// SIMATIC S7-200 project (STEP 7-Micro/WIN), CPU 221 REL 01.10

SYMBOL_TABLE USR1
First_Scan_On    SM0.1    // This bit is on for the first scan cycle only.
Edge_Up          MW1      // The number of positive transitions at input I0.0 is stored in MW1.
Edge_Down        MW3      // The number of negative transitions at input I0.1 is stored in MW3.
END_SYMBOL_TABLE

ORGANIZATION_BLOCK MAIN:OB1
TITLE=
//  题目：检测输入信号的边沿
// ***概述***
// 本例程序用来说明如何用S7-200的检测边沿指令来检测简单信号的变化。在这个过程中，
// 用上升和下降来区分信号边沿，上升沿指信号由“0”变为“1”，下降沿指信
// 号由“1”变为“0”。逻辑“1”表示输入上有电压，“0”表示输入上无电压。
// 程序用2个存储字分别累计输入I0.0上升沿数目以及输入I0.1下降沿数目。
// ***程序和注释***
// 程序例用输入I0.0和EU（上升沿）指令来判定上升沿变化是否发生，也就是说，
// 信号由“0”变为“1”。如果一个上升沿变化发生了，那么存储字MW1的值增加1
// ED(下降沿)指令用来计数输入I0.1的下降沿，用存储字MW3来计数。如果某一个
// 存储字计数达到127，那么该存储字被重新置为0。注意MB2是存储字MW1的低字节，
// MB1为高字节。同样的，MB4为存储字MW3的低字节，MB3为高字节。
// 标题：检测边沿
// 
BEGIN
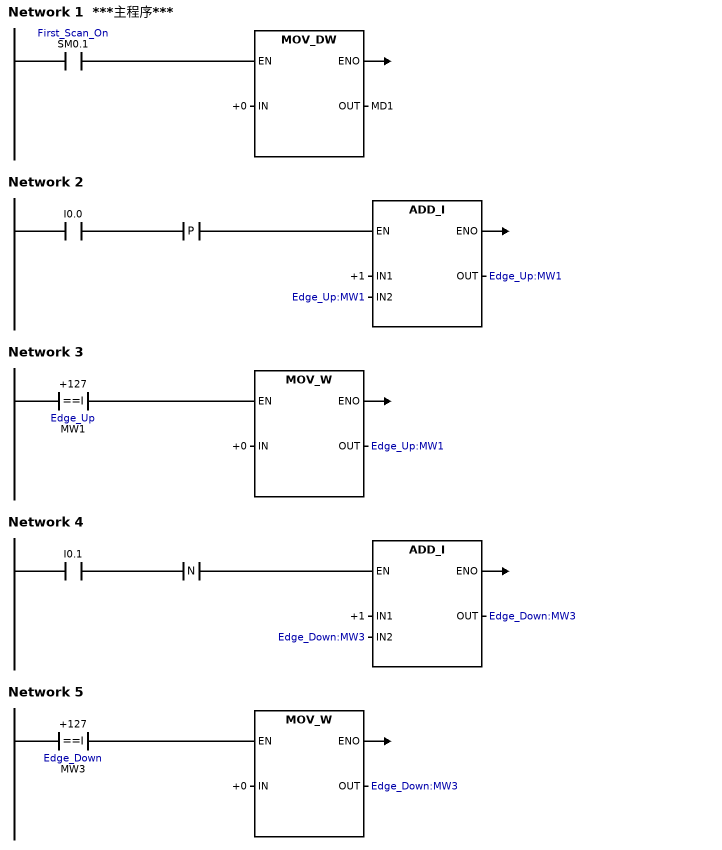
Network 1 // ***主程序***	
// 仅在第一次扫描时 SM0.1=1。
// 把存储器双字 MD1置0
LD     First_Scan_On:SM0.1
MOVD   +0, MD1
Network 2
// 输入信号 I0.0.
// 上升沿
// 存储字MW1的值加1
LD     I0.0
EU
+I     +1, Edge_Up:MW1
Network 3
// 如果累计127个上升沿变化（或某个指定的值）
// 则将存储字MW1置0
LDW=   +127, Edge_Up:MW1
MOVW   +0, Edge_Up:MW1
Network 4
// 输入信号 I0.0.
// 下降沿
// 下降沿变化，使存储字MW3的值加1
LD     I0.1
ED
+I     +1, Edge_Down:MW3
Network 5
// 如果累计127个下降沿变化（或某个指定的值）
//则将存储字MW3置0
LDW=   +127, Edge_Down:MW3
MOVW   +0, Edge_Down:MW3
Network 6 //  主程序结束
// MEND				
// 
END_ORGANIZATION_BLOCK
